PROGRAM main
VAR
	Auto_Mode_En : bool;
	START_CMD0 : Start_CMD;
	Hand_Mode_En : bool;
	Auto_Relay : bool;
	Run_CMD : bool;
	Hand_Relay : bool;
	STA_Butt : bool;
	STP_Butt : bool;
	Run_Perm : bool;
	Auto_Req : bool;
	VFD_Fault_Latched : bool;
	VFD_Fault : bool;
	Press_Fault_Latched : bool;
	High_Press : bool;
	Reset_Cmd : bool;
	Reset_Butt : bool;
	Hand_Req : bool;
	Auto_Inhib : bool;
	Tank_Lvl_High : bool;
	Above_Low_Lvl : bool;
	High_Lvl_Sw : bool;
	Low_Lvl_Sw : bool;
END_VAR

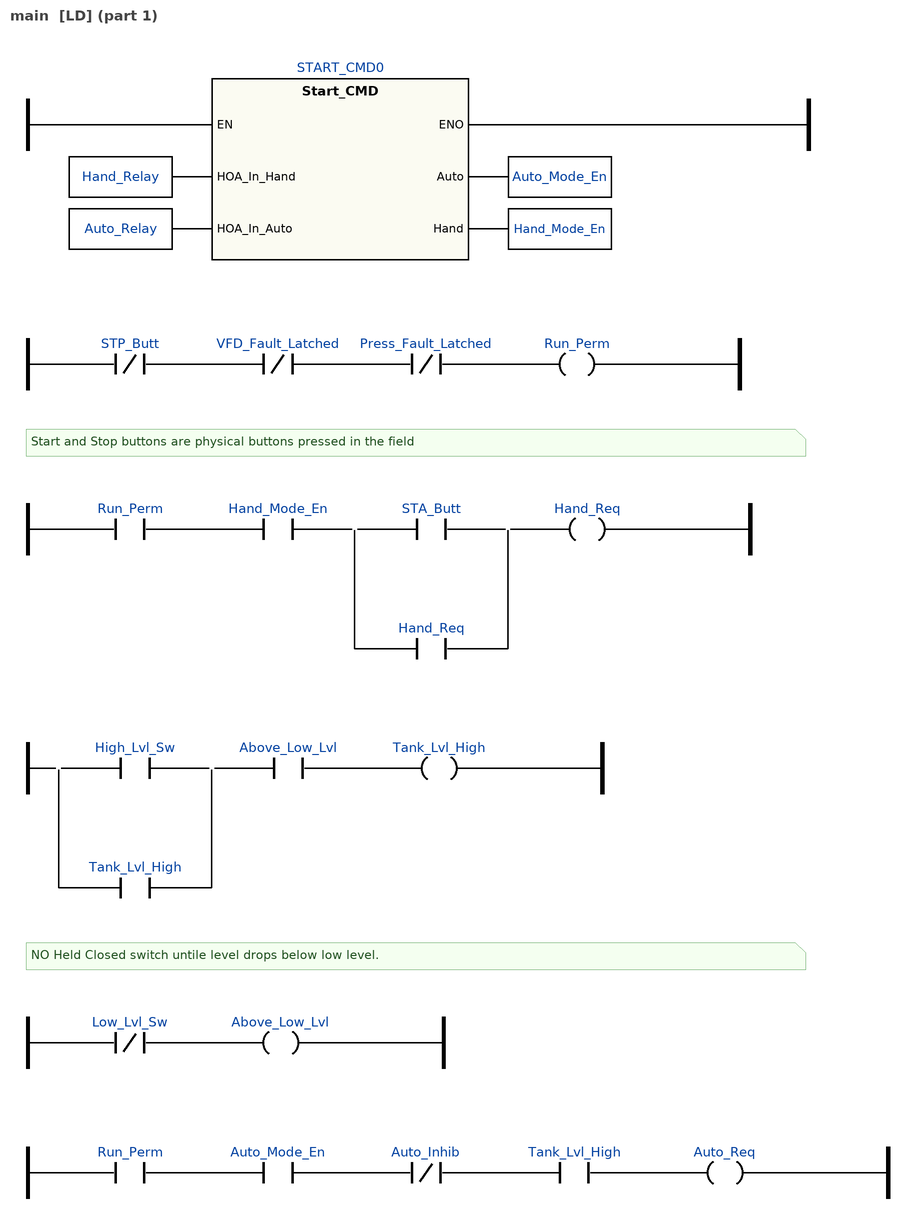
(* LD diagram, written out as Structured Text *)
START_CMD0(HOA_In_Hand := Hand_Relay, HOA_In_Auto := Auto_Relay);
Auto_Mode_En := START_CMD0.Auto;
Hand_Mode_En := START_CMD0.Hand;
Run_Perm := NOT STP_Butt AND NOT VFD_Fault_Latched AND NOT Press_Fault_Latched;
(* Start and Stop buttons are physical buttons pressed in the field *)
Hand_Req := Run_Perm AND Hand_Mode_En AND (STA_Butt OR Hand_Req);
Tank_Lvl_High := (High_Lvl_Sw OR Tank_Lvl_High) AND Above_Low_Lvl;
(* NO Held Closed switch untile level drops below low level. *)
Above_Low_Lvl := NOT Low_Lvl_Sw;
Auto_Req := Run_Perm AND Auto_Mode_En AND NOT Auto_Inhib AND Tank_Lvl_High;
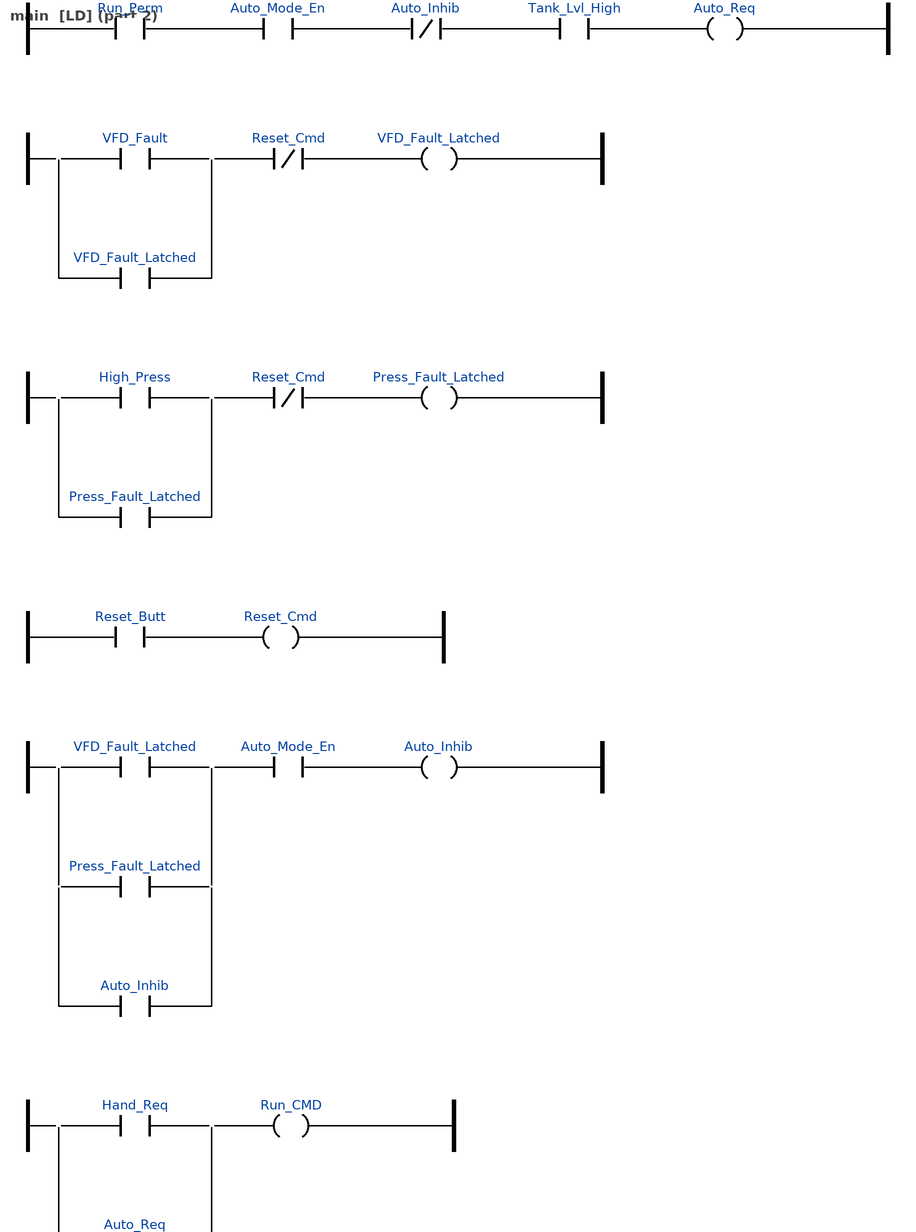
VFD_Fault_Latched := (VFD_Fault OR VFD_Fault_Latched) AND NOT Reset_Cmd;
Press_Fault_Latched := (High_Press OR Press_Fault_Latched) AND NOT Reset_Cmd;
Reset_Cmd := Reset_Butt;
Auto_Inhib := (VFD_Fault_Latched OR Press_Fault_Latched OR Auto_Inhib) AND Auto_Mode_En;
Run_CMD := Hand_Req OR Auto_Req;
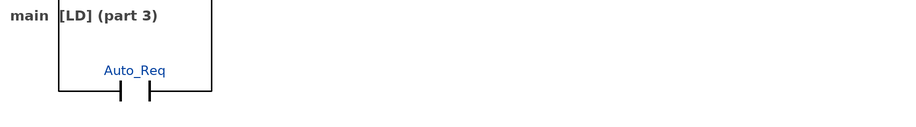
END_PROGRAM
